TYPE PLCStruct :
STRUCT
	intVal : INT;
 	dintVal    : DINT;
	byteVal    : SINT;
	lrealVal  : LREAL;
	realVal  : REAL;
END_STRUCT
END_TYPE

(* stored: Version 1.1.0.1, ProductVersion 3.1.4024.9
   DUT PLCStruct: Id {908de95f-fd92-4bc3-8745-5b095fa9f454} *)
